// TIA Portal V18 export
// export: Created 2026-01-09T11:31:52.2336406Z, ExportSetting WithDefaults, DisplayName Totally Integrated Automation Portal, DisplayVersion V18 Update 5, DisplayName TIA Portal Openness, DisplayVersion V18 Update 5, DisplayName TIA Portal Teamcenter Gateway, DisplayVersion V18, DisplayName TIA Portal Version Control Interface, DisplayVersion V18, DisplayName SINAMICS Startdrive Advanced, DisplayVersion V18 SP2 Update 1, DisplayName SINAMICS Startdrive G110M, G120, G120C, G120D, G120P, G115D, DisplayVersion V18 SP2 Update 1, DisplayName SINAMICS Startdrive G130, G150, S120, S150, SINAMICS MV, S210, G220, S200, DisplayVersion V18 SP2 Update 1, DisplayName STEP 7 Professional, DisplayVersion V18 Update 5, DisplayName STEP 7 Safety, DisplayVersion V18, DisplayName WinCC Professional, DisplayVersion V18 Update 5
TagTable "ProcessData_Buffet"
  AutoProcessData_Buffer_DataBuffer_1 : ProcessData  (PLC tag AutoProcessData_Buffer.DataBuffer_1, CPU S71500-2PN_TP700, 500 ms)
    TagStructureMember "PartStatus"
    TagStructureMember "PartSNGCode"
    TagStructureMember "PartRemoveFlag"
    TagStructureMember "Spare1"
    TagStructureMember "Spare2"
    TagStructureMember "Spare3"
    TagStructureMember "Spare4"
    TagStructureMember "Spare5"
    TagStructureMember "Spare6"
    TagStructureMember "Spare7"
    TagStructureMember "Spare8"
    TagStructureMember "Spare9"
    TagStructureMember "Spare10"
    TagStructureMember "Spare11"
    TagStructureMember "Spare12"
    TagStructureMember "Spare13"
    TagStructureMember "Spare14"
    TagStructureMember "Spare15"
    TagStructureMember "ShaftCode"
    TagStructureMember "RingCode_1"
    TagStructureMember "Code_1"
    TagStructureMember "RingCode_2"
    TagStructureMember "TableCode_1"
    TagStructureMember "TableCode_2"
    TagStructureMember "Press1Program"
    TagStructureMember "Press1FinalPosition"
    TagStructureMember "Press1FinalForce"
    TagStructureMember "Press2Program"
    TagStructureMember "Press2FinalPosition"
    TagStructureMember "Press2FinalForce"
    TagStructureMember "IV3_ShaftCheckResult"
    TagStructureMember "IV3_ShaftScore_1"
    TagStructureMember "IV3_ShaftScore_2"
    TagStructureMember "IV3_ShaftScore_3"
    TagStructureMember "IV3_ShaftScore_4"
    TagStructureMember "IV3_MagnetCheckResult"
    TagStructureMember "IV3_MagnetScore"
    TagStructureMember "Spare_3"
      TagArrayMember "[0]"
      TagArrayMember "[1]"
      TagArrayMember "[2]"
      TagArrayMember "[3]"
      TagArrayMember "[4]"
      TagArrayMember "[5]"
      TagArrayMember "[6]"
      TagArrayMember "[7]"
      TagArrayMember "[8]"
      TagArrayMember "[9]"
      TagArrayMember "[10]"
      TagArrayMember "[11]"
      TagArrayMember "[12]"
      TagArrayMember "[13]"
      TagArrayMember "[14]"
      TagArrayMember "[15]"
      TagArrayMember "[16]"
      TagArrayMember "[17]"
      TagArrayMember "[18]"
      TagArrayMember "[19]"
      TagArrayMember "[20]"
      TagArrayMember "[21]"
      TagArrayMember "[22]"
      TagArrayMember "[23]"
      TagArrayMember "[24]"
      TagArrayMember "[25]"
      TagArrayMember "[26]"
      TagArrayMember "[27]"
      TagArrayMember "[28]"
      TagArrayMember "[29]"
      TagArrayMember "[30]"
      TagArrayMember "[31]"
      TagArrayMember "[32]"
      TagArrayMember "[33]"
      TagArrayMember "[34]"
      TagArrayMember "[35]"
      TagArrayMember "[36]"
      TagArrayMember "[37]"
      TagArrayMember "[38]"
      TagArrayMember "[39]"
      TagArrayMember "[40]"
      TagArrayMember "[41]"
      TagArrayMember "[42]"
      TagArrayMember "[43]"
      TagArrayMember "[44]"
      TagArrayMember "[45]"
      TagArrayMember "[46]"
      TagArrayMember "[47]"
      TagArrayMember "[48]"
      TagArrayMember "[49]"
      TagArrayMember "[50]"
      TagArrayMember "[51]"
      TagArrayMember "[52]"
      TagArrayMember "[53]"
      TagArrayMember "[54]"
      TagArrayMember "[55]"
      TagArrayMember "[56]"
      TagArrayMember "[57]"
      TagArrayMember "[58]"
      TagArrayMember "[59]"
      TagArrayMember "[60]"
      TagArrayMember "[61]"
      TagArrayMember "[62]"
      TagArrayMember "[63]"
      TagArrayMember "[64]"
      TagArrayMember "[65]"
      TagArrayMember "[66]"
      TagArrayMember "[67]"
      TagArrayMember "[68]"
      TagArrayMember "[69]"
      TagArrayMember "[70]"
      TagArrayMember "[71]"
      TagArrayMember "[72]"
      TagArrayMember "[73]"
      TagArrayMember "[74]"
      TagArrayMember "[75]"
      TagArrayMember "[76]"
      TagArrayMember "[77]"
      TagArrayMember "[78]"
      TagArrayMember "[79]"
      TagArrayMember "[80]"
      TagArrayMember "[81]"
      TagArrayMember "[82]"
      TagArrayMember "[83]"
      TagArrayMember "[84]"
      TagArrayMember "[85]"
      TagArrayMember "[86]"
      TagArrayMember "[87]"
      TagArrayMember "[88]"
      TagArrayMember "[89]"
  AutoProcessData_Buffer_DataBuffer_2 : ProcessData  (PLC tag AutoProcessData_Buffer.DataBuffer_2, CPU S71500-2PN_TP700, 500 ms)
    TagStructureMember "PartStatus"
    TagStructureMember "PartSNGCode"
    TagStructureMember "PartRemoveFlag"
    TagStructureMember "Spare1"
    TagStructureMember "Spare2"
    TagStructureMember "Spare3"
    TagStructureMember "Spare4"
    TagStructureMember "Spare5"
    TagStructureMember "Spare6"
    TagStructureMember "Spare7"
    TagStructureMember "Spare8"
    TagStructureMember "Spare9"
    TagStructureMember "Spare10"
    TagStructureMember "Spare11"
    TagStructureMember "Spare12"
    TagStructureMember "Spare13"
    TagStructureMember "Spare14"
    TagStructureMember "Spare15"
    TagStructureMember "ShaftCode"
    TagStructureMember "RingCode_1"
    TagStructureMember "Code_1"
    TagStructureMember "RingCode_2"
    TagStructureMember "TableCode_1"
    TagStructureMember "TableCode_2"
    TagStructureMember "Press1Program"
    TagStructureMember "Press1FinalPosition"
    TagStructureMember "Press1FinalForce"
    TagStructureMember "Press2Program"
    TagStructureMember "Press2FinalPosition"
    TagStructureMember "Press2FinalForce"
    TagStructureMember "IV3_ShaftCheckResult"
    TagStructureMember "IV3_ShaftScore_1"
    TagStructureMember "IV3_ShaftScore_2"
    TagStructureMember "IV3_ShaftScore_3"
    TagStructureMember "IV3_ShaftScore_4"
    TagStructureMember "IV3_MagnetCheckResult"
    TagStructureMember "IV3_MagnetScore"
    TagStructureMember "Spare_3"
      TagArrayMember "[0]"
      TagArrayMember "[1]"
      TagArrayMember "[2]"
      TagArrayMember "[3]"
      TagArrayMember "[4]"
      TagArrayMember "[5]"
      TagArrayMember "[6]"
      TagArrayMember "[7]"
      TagArrayMember "[8]"
      TagArrayMember "[9]"
      TagArrayMember "[10]"
      TagArrayMember "[11]"
      TagArrayMember "[12]"
      TagArrayMember "[13]"
      TagArrayMember "[14]"
      TagArrayMember "[15]"
      TagArrayMember "[16]"
      TagArrayMember "[17]"
      TagArrayMember "[18]"
      TagArrayMember "[19]"
      TagArrayMember "[20]"
      TagArrayMember "[21]"
      TagArrayMember "[22]"
      TagArrayMember "[23]"
      TagArrayMember "[24]"
      TagArrayMember "[25]"
      TagArrayMember "[26]"
      TagArrayMember "[27]"
      TagArrayMember "[28]"
      TagArrayMember "[29]"
      TagArrayMember "[30]"
      TagArrayMember "[31]"
      TagArrayMember "[32]"
      TagArrayMember "[33]"
      TagArrayMember "[34]"
      TagArrayMember "[35]"
      TagArrayMember "[36]"
      TagArrayMember "[37]"
      TagArrayMember "[38]"
      TagArrayMember "[39]"
      TagArrayMember "[40]"
      TagArrayMember "[41]"
      TagArrayMember "[42]"
      TagArrayMember "[43]"
      TagArrayMember "[44]"
      TagArrayMember "[45]"
      TagArrayMember "[46]"
      TagArrayMember "[47]"
      TagArrayMember "[48]"
      TagArrayMember "[49]"
      TagArrayMember "[50]"
      TagArrayMember "[51]"
      TagArrayMember "[52]"
      TagArrayMember "[53]"
      TagArrayMember "[54]"
      TagArrayMember "[55]"
      TagArrayMember "[56]"
      TagArrayMember "[57]"
      TagArrayMember "[58]"
      TagArrayMember "[59]"
      TagArrayMember "[60]"
      TagArrayMember "[61]"
      TagArrayMember "[62]"
      TagArrayMember "[63]"
      TagArrayMember "[64]"
      TagArrayMember "[65]"
      TagArrayMember "[66]"
      TagArrayMember "[67]"
      TagArrayMember "[68]"
      TagArrayMember "[69]"
      TagArrayMember "[70]"
      TagArrayMember "[71]"
      TagArrayMember "[72]"
      TagArrayMember "[73]"
      TagArrayMember "[74]"
      TagArrayMember "[75]"
      TagArrayMember "[76]"
      TagArrayMember "[77]"
      TagArrayMember "[78]"
      TagArrayMember "[79]"
      TagArrayMember "[80]"
      TagArrayMember "[81]"
      TagArrayMember "[82]"
      TagArrayMember "[83]"
      TagArrayMember "[84]"
      TagArrayMember "[85]"
      TagArrayMember "[86]"
      TagArrayMember "[87]"
      TagArrayMember "[88]"
      TagArrayMember "[89]"
  AutoProcessData_Buffer_DataBuffer_3 : ProcessData  (PLC tag AutoProcessData_Buffer.DataBuffer_3, CPU S71500-2PN_TP700, 500 ms)
    TagStructureMember "PartStatus"
    TagStructureMember "PartSNGCode"
    TagStructureMember "PartRemoveFlag"
    TagStructureMember "Spare1"
    TagStructureMember "Spare2"
    TagStructureMember "Spare3"
    TagStructureMember "Spare4"
    TagStructureMember "Spare5"
    TagStructureMember "Spare6"
    TagStructureMember "Spare7"
    TagStructureMember "Spare8"
    TagStructureMember "Spare9"
    TagStructureMember "Spare10"
    TagStructureMember "Spare11"
    TagStructureMember "Spare12"
    TagStructureMember "Spare13"
    TagStructureMember "Spare14"
    TagStructureMember "Spare15"
    TagStructureMember "ShaftCode"
    TagStructureMember "RingCode_1"
    TagStructureMember "Code_1"
    TagStructureMember "RingCode_2"
    TagStructureMember "TableCode_1"
    TagStructureMember "TableCode_2"
    TagStructureMember "Press1Program"
    TagStructureMember "Press1FinalPosition"
    TagStructureMember "Press1FinalForce"
    TagStructureMember "Press2Program"
    TagStructureMember "Press2FinalPosition"
    TagStructureMember "Press2FinalForce"
    TagStructureMember "IV3_ShaftCheckResult"
    TagStructureMember "IV3_ShaftScore_1"
    TagStructureMember "IV3_ShaftScore_2"
    TagStructureMember "IV3_ShaftScore_3"
    TagStructureMember "IV3_ShaftScore_4"
    TagStructureMember "IV3_MagnetCheckResult"
    TagStructureMember "IV3_MagnetScore"
    TagStructureMember "Spare_3"
      TagArrayMember "[0]"
      TagArrayMember "[1]"
      TagArrayMember "[2]"
      TagArrayMember "[3]"
      TagArrayMember "[4]"
      TagArrayMember "[5]"
      TagArrayMember "[6]"
      TagArrayMember "[7]"
      TagArrayMember "[8]"
      TagArrayMember "[9]"
      TagArrayMember "[10]"
      TagArrayMember "[11]"
      TagArrayMember "[12]"
      TagArrayMember "[13]"
      TagArrayMember "[14]"
      TagArrayMember "[15]"
      TagArrayMember "[16]"
      TagArrayMember "[17]"
      TagArrayMember "[18]"
      TagArrayMember "[19]"
      TagArrayMember "[20]"
      TagArrayMember "[21]"
      TagArrayMember "[22]"
      TagArrayMember "[23]"
      TagArrayMember "[24]"
      TagArrayMember "[25]"
      TagArrayMember "[26]"
      TagArrayMember "[27]"
      TagArrayMember "[28]"
      TagArrayMember "[29]"
      TagArrayMember "[30]"
      TagArrayMember "[31]"
      TagArrayMember "[32]"
      TagArrayMember "[33]"
      TagArrayMember "[34]"
      TagArrayMember "[35]"
      TagArrayMember "[36]"
      TagArrayMember "[37]"
      TagArrayMember "[38]"
      TagArrayMember "[39]"
      TagArrayMember "[40]"
      TagArrayMember "[41]"
      TagArrayMember "[42]"
      TagArrayMember "[43]"
      TagArrayMember "[44]"
      TagArrayMember "[45]"
      TagArrayMember "[46]"
      TagArrayMember "[47]"
      TagArrayMember "[48]"
      TagArrayMember "[49]"
      TagArrayMember "[50]"
      TagArrayMember "[51]"
      TagArrayMember "[52]"
      TagArrayMember "[53]"
      TagArrayMember "[54]"
      TagArrayMember "[55]"
      TagArrayMember "[56]"
      TagArrayMember "[57]"
      TagArrayMember "[58]"
      TagArrayMember "[59]"
      TagArrayMember "[60]"
      TagArrayMember "[61]"
      TagArrayMember "[62]"
      TagArrayMember "[63]"
      TagArrayMember "[64]"
      TagArrayMember "[65]"
      TagArrayMember "[66]"
      TagArrayMember "[67]"
      TagArrayMember "[68]"
      TagArrayMember "[69]"
      TagArrayMember "[70]"
      TagArrayMember "[71]"
      TagArrayMember "[72]"
      TagArrayMember "[73]"
      TagArrayMember "[74]"
      TagArrayMember "[75]"
      TagArrayMember "[76]"
      TagArrayMember "[77]"
      TagArrayMember "[78]"
      TagArrayMember "[79]"
      TagArrayMember "[80]"
      TagArrayMember "[81]"
      TagArrayMember "[82]"
      TagArrayMember "[83]"
      TagArrayMember "[84]"
      TagArrayMember "[85]"
      TagArrayMember "[86]"
      TagArrayMember "[87]"
      TagArrayMember "[88]"
      TagArrayMember "[89]"
  AutoProcessData_Buffer_DataBuffer_4 : ProcessData  (PLC tag AutoProcessData_Buffer.DataBuffer_4, CPU S71500-2PN_TP700, 500 ms)
    TagStructureMember "PartStatus"
    TagStructureMember "PartSNGCode"
    TagStructureMember "PartRemoveFlag"
    TagStructureMember "Spare1"
    TagStructureMember "Spare2"
    TagStructureMember "Spare3"
    TagStructureMember "Spare4"
    TagStructureMember "Spare5"
    TagStructureMember "Spare6"
    TagStructureMember "Spare7"
    TagStructureMember "Spare8"
    TagStructureMember "Spare9"
    TagStructureMember "Spare10"
    TagStructureMember "Spare11"
    TagStructureMember "Spare12"
    TagStructureMember "Spare13"
    TagStructureMember "Spare14"
    TagStructureMember "Spare15"
    TagStructureMember "ShaftCode"
    TagStructureMember "RingCode_1"
    TagStructureMember "Code_1"
    TagStructureMember "RingCode_2"
    TagStructureMember "TableCode_1"
    TagStructureMember "TableCode_2"
    TagStructureMember "Press1Program"
    TagStructureMember "Press1FinalPosition"
    TagStructureMember "Press1FinalForce"
    TagStructureMember "Press2Program"
    TagStructureMember "Press2FinalPosition"
    TagStructureMember "Press2FinalForce"
    TagStructureMember "IV3_ShaftCheckResult"
    TagStructureMember "IV3_ShaftScore_1"
    TagStructureMember "IV3_ShaftScore_2"
    TagStructureMember "IV3_ShaftScore_3"
    TagStructureMember "IV3_ShaftScore_4"
    TagStructureMember "IV3_MagnetCheckResult"
    TagStructureMember "IV3_MagnetScore"
    TagStructureMember "Spare_3"
      TagArrayMember "[0]"
      TagArrayMember "[1]"
      TagArrayMember "[2]"
      TagArrayMember "[3]"
      TagArrayMember "[4]"
      TagArrayMember "[5]"
      TagArrayMember "[6]"
      TagArrayMember "[7]"
      TagArrayMember "[8]"
      TagArrayMember "[9]"
      TagArrayMember "[10]"
      TagArrayMember "[11]"
      TagArrayMember "[12]"
      TagArrayMember "[13]"
      TagArrayMember "[14]"
      TagArrayMember "[15]"
      TagArrayMember "[16]"
      TagArrayMember "[17]"
      TagArrayMember "[18]"
      TagArrayMember "[19]"
      TagArrayMember "[20]"
      TagArrayMember "[21]"
      TagArrayMember "[22]"
      TagArrayMember "[23]"
      TagArrayMember "[24]"
      TagArrayMember "[25]"
      TagArrayMember "[26]"
      TagArrayMember "[27]"
      TagArrayMember "[28]"
      TagArrayMember "[29]"
      TagArrayMember "[30]"
      TagArrayMember "[31]"
      TagArrayMember "[32]"
      TagArrayMember "[33]"
      TagArrayMember "[34]"
      TagArrayMember "[35]"
      TagArrayMember "[36]"
      TagArrayMember "[37]"
      TagArrayMember "[38]"
      TagArrayMember "[39]"
      TagArrayMember "[40]"
      TagArrayMember "[41]"
      TagArrayMember "[42]"
      TagArrayMember "[43]"
      TagArrayMember "[44]"
      TagArrayMember "[45]"
      TagArrayMember "[46]"
      TagArrayMember "[47]"
      TagArrayMember "[48]"
      TagArrayMember "[49]"
      TagArrayMember "[50]"
      TagArrayMember "[51]"
      TagArrayMember "[52]"
      TagArrayMember "[53]"
      TagArrayMember "[54]"
      TagArrayMember "[55]"
      TagArrayMember "[56]"
      TagArrayMember "[57]"
      TagArrayMember "[58]"
      TagArrayMember "[59]"
      TagArrayMember "[60]"
      TagArrayMember "[61]"
      TagArrayMember "[62]"
      TagArrayMember "[63]"
      TagArrayMember "[64]"
      TagArrayMember "[65]"
      TagArrayMember "[66]"
      TagArrayMember "[67]"
      TagArrayMember "[68]"
      TagArrayMember "[69]"
      TagArrayMember "[70]"
      TagArrayMember "[71]"
      TagArrayMember "[72]"
      TagArrayMember "[73]"
      TagArrayMember "[74]"
      TagArrayMember "[75]"
      TagArrayMember "[76]"
      TagArrayMember "[77]"
      TagArrayMember "[78]"
      TagArrayMember "[79]"
      TagArrayMember "[80]"
      TagArrayMember "[81]"
      TagArrayMember "[82]"
      TagArrayMember "[83]"
      TagArrayMember "[84]"
      TagArrayMember "[85]"
      TagArrayMember "[86]"
      TagArrayMember "[87]"
      TagArrayMember "[88]"
      TagArrayMember "[89]"
  AutoProcessData_Buffer_DataBuffer_5 : ProcessData  (PLC tag AutoProcessData_Buffer.DataBuffer_5, CPU S71500-2PN_TP700, 500 ms)
    TagStructureMember "PartStatus"
    TagStructureMember "PartSNGCode"
    TagStructureMember "PartRemoveFlag"
    TagStructureMember "Spare1"
    TagStructureMember "Spare2"
    TagStructureMember "Spare3"
    TagStructureMember "Spare4"
    TagStructureMember "Spare5"
    TagStructureMember "Spare6"
    TagStructureMember "Spare7"
    TagStructureMember "Spare8"
    TagStructureMember "Spare9"
    TagStructureMember "Spare10"
    TagStructureMember "Spare11"
    TagStructureMember "Spare12"
    TagStructureMember "Spare13"
    TagStructureMember "Spare14"
    TagStructureMember "Spare15"
    TagStructureMember "ShaftCode"
    TagStructureMember "RingCode_1"
    TagStructureMember "Code_1"
    TagStructureMember "RingCode_2"
    TagStructureMember "TableCode_1"
    TagStructureMember "TableCode_2"
    TagStructureMember "Press1Program"
    TagStructureMember "Press1FinalPosition"
    TagStructureMember "Press1FinalForce"
    TagStructureMember "Press2Program"
    TagStructureMember "Press2FinalPosition"
    TagStructureMember "Press2FinalForce"
    TagStructureMember "IV3_ShaftCheckResult"
    TagStructureMember "IV3_ShaftScore_1"
    TagStructureMember "IV3_ShaftScore_2"
    TagStructureMember "IV3_ShaftScore_3"
    TagStructureMember "IV3_ShaftScore_4"
    TagStructureMember "IV3_MagnetCheckResult"
    TagStructureMember "IV3_MagnetScore"
    TagStructureMember "Spare_3"
      TagArrayMember "[0]"
      TagArrayMember "[1]"
      TagArrayMember "[2]"
      TagArrayMember "[3]"
      TagArrayMember "[4]"
      TagArrayMember "[5]"
      TagArrayMember "[6]"
      TagArrayMember "[7]"
      TagArrayMember "[8]"
      TagArrayMember "[9]"
      TagArrayMember "[10]"
      TagArrayMember "[11]"
      TagArrayMember "[12]"
      TagArrayMember "[13]"
      TagArrayMember "[14]"
      TagArrayMember "[15]"
      TagArrayMember "[16]"
      TagArrayMember "[17]"
      TagArrayMember "[18]"
      TagArrayMember "[19]"
      TagArrayMember "[20]"
      TagArrayMember "[21]"
      TagArrayMember "[22]"
      TagArrayMember "[23]"
      TagArrayMember "[24]"
      TagArrayMember "[25]"
      TagArrayMember "[26]"
      TagArrayMember "[27]"
      TagArrayMember "[28]"
      TagArrayMember "[29]"
      TagArrayMember "[30]"
      TagArrayMember "[31]"
      TagArrayMember "[32]"
      TagArrayMember "[33]"
      TagArrayMember "[34]"
      TagArrayMember "[35]"
      TagArrayMember "[36]"
      TagArrayMember "[37]"
      TagArrayMember "[38]"
      TagArrayMember "[39]"
      TagArrayMember "[40]"
      TagArrayMember "[41]"
      TagArrayMember "[42]"
      TagArrayMember "[43]"
      TagArrayMember "[44]"
      TagArrayMember "[45]"
      TagArrayMember "[46]"
      TagArrayMember "[47]"
      TagArrayMember "[48]"
      TagArrayMember "[49]"
      TagArrayMember "[50]"
      TagArrayMember "[51]"
      TagArrayMember "[52]"
      TagArrayMember "[53]"
      TagArrayMember "[54]"
      TagArrayMember "[55]"
      TagArrayMember "[56]"
      TagArrayMember "[57]"
      TagArrayMember "[58]"
      TagArrayMember "[59]"
      TagArrayMember "[60]"
      TagArrayMember "[61]"
      TagArrayMember "[62]"
      TagArrayMember "[63]"
      TagArrayMember "[64]"
      TagArrayMember "[65]"
      TagArrayMember "[66]"
      TagArrayMember "[67]"
      TagArrayMember "[68]"
      TagArrayMember "[69]"
      TagArrayMember "[70]"
      TagArrayMember "[71]"
      TagArrayMember "[72]"
      TagArrayMember "[73]"
      TagArrayMember "[74]"
      TagArrayMember "[75]"
      TagArrayMember "[76]"
      TagArrayMember "[77]"
      TagArrayMember "[78]"
      TagArrayMember "[79]"
      TagArrayMember "[80]"
      TagArrayMember "[81]"
      TagArrayMember "[82]"
      TagArrayMember "[83]"
      TagArrayMember "[84]"
      TagArrayMember "[85]"
      TagArrayMember "[86]"
      TagArrayMember "[87]"
      TagArrayMember "[88]"
      TagArrayMember "[89]"
  AutoProcessData_Buffer_DataBuffer_6 : ProcessData  (PLC tag AutoProcessData_Buffer.DataBuffer_6, CPU S71500-2PN_TP700, 500 ms)
    TagStructureMember "PartStatus"
    TagStructureMember "PartSNGCode"
    TagStructureMember "PartRemoveFlag"
    TagStructureMember "Spare1"
    TagStructureMember "Spare2"
    TagStructureMember "Spare3"
    TagStructureMember "Spare4"
    TagStructureMember "Spare5"
    TagStructureMember "Spare6"
    TagStructureMember "Spare7"
    TagStructureMember "Spare8"
    TagStructureMember "Spare9"
    TagStructureMember "Spare10"
    TagStructureMember "Spare11"
    TagStructureMember "Spare12"
    TagStructureMember "Spare13"
    TagStructureMember "Spare14"
    TagStructureMember "Spare15"
    TagStructureMember "ShaftCode"
    TagStructureMember "RingCode_1"
    TagStructureMember "Code_1"
    TagStructureMember "RingCode_2"
    TagStructureMember "TableCode_1"
    TagStructureMember "TableCode_2"
    TagStructureMember "Press1Program"
    TagStructureMember "Press1FinalPosition"
    TagStructureMember "Press1FinalForce"
    TagStructureMember "Press2Program"
    TagStructureMember "Press2FinalPosition"
    TagStructureMember "Press2FinalForce"
    TagStructureMember "IV3_ShaftCheckResult"
    TagStructureMember "IV3_ShaftScore_1"
    TagStructureMember "IV3_ShaftScore_2"
    TagStructureMember "IV3_ShaftScore_3"
    TagStructureMember "IV3_ShaftScore_4"
    TagStructureMember "IV3_MagnetCheckResult"
    TagStructureMember "IV3_MagnetScore"
    TagStructureMember "Spare_3"
      TagArrayMember "[0]"
      TagArrayMember "[1]"
      TagArrayMember "[2]"
      TagArrayMember "[3]"
      TagArrayMember "[4]"
      TagArrayMember "[5]"
      TagArrayMember "[6]"
      TagArrayMember "[7]"
      TagArrayMember "[8]"
      TagArrayMember "[9]"
      TagArrayMember "[10]"
      TagArrayMember "[11]"
      TagArrayMember "[12]"
      TagArrayMember "[13]"
      TagArrayMember "[14]"
      TagArrayMember "[15]"
      TagArrayMember "[16]"
      TagArrayMember "[17]"
      TagArrayMember "[18]"
      TagArrayMember "[19]"
      TagArrayMember "[20]"
      TagArrayMember "[21]"
      TagArrayMember "[22]"
      TagArrayMember "[23]"
      TagArrayMember "[24]"
      TagArrayMember "[25]"
      TagArrayMember "[26]"
      TagArrayMember "[27]"
      TagArrayMember "[28]"
      TagArrayMember "[29]"
      TagArrayMember "[30]"
      TagArrayMember "[31]"
      TagArrayMember "[32]"
      TagArrayMember "[33]"
      TagArrayMember "[34]"
      TagArrayMember "[35]"
      TagArrayMember "[36]"
      TagArrayMember "[37]"
      TagArrayMember "[38]"
      TagArrayMember "[39]"
      TagArrayMember "[40]"
      TagArrayMember "[41]"
      TagArrayMember "[42]"
      TagArrayMember "[43]"
      TagArrayMember "[44]"
      TagArrayMember "[45]"
      TagArrayMember "[46]"
      TagArrayMember "[47]"
      TagArrayMember "[48]"
      TagArrayMember "[49]"
      TagArrayMember "[50]"
      TagArrayMember "[51]"
      TagArrayMember "[52]"
      TagArrayMember "[53]"
      TagArrayMember "[54]"
      TagArrayMember "[55]"
      TagArrayMember "[56]"
      TagArrayMember "[57]"
      TagArrayMember "[58]"
      TagArrayMember "[59]"
      TagArrayMember "[60]"
      TagArrayMember "[61]"
      TagArrayMember "[62]"
      TagArrayMember "[63]"
      TagArrayMember "[64]"
      TagArrayMember "[65]"
      TagArrayMember "[66]"
      TagArrayMember "[67]"
      TagArrayMember "[68]"
      TagArrayMember "[69]"
      TagArrayMember "[70]"
      TagArrayMember "[71]"
      TagArrayMember "[72]"
      TagArrayMember "[73]"
      TagArrayMember "[74]"
      TagArrayMember "[75]"
      TagArrayMember "[76]"
      TagArrayMember "[77]"
      TagArrayMember "[78]"
      TagArrayMember "[79]"
      TagArrayMember "[80]"
      TagArrayMember "[81]"
      TagArrayMember "[82]"
      TagArrayMember "[83]"
      TagArrayMember "[84]"
      TagArrayMember "[85]"
      TagArrayMember "[86]"
      TagArrayMember "[87]"
      TagArrayMember "[88]"
      TagArrayMember "[89]"
  AutoProcessData_Buffer_SelectButton : Int  (PLC tag AutoProcessData_Buffer.SelectButton, CPU S71500-2PN_TP700, 500 ms)
